FUNCTION_BLOCK AE_DEMUX_5 (* AE demultiplexor (generic FB) *)
  (* Standard: 61499-2; Description: Copyright (c) 2026 HR Agrartechnik GmbH This program and the accompanying materials are made available under the terms of the Eclipse Public License 2.0 which is available at https://www.eclipse.org/legal/epl-2.0/ SPDX-License-Identifier: EPL-2.0 *)
  (* Version 1.0, 2026-05-28, Franz Höpfinger, HR Agrartechnik GmbH *)
  PACKAGE adapter::selection::unidirectional;
  IMPORT eclipse4diac::core::TypeHash;
  {SET_ATTRIBUTE(eclipse4diac::core::GenericClassName, 'GEN_AE_DEMUX')}
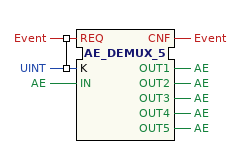
  EVENT_INPUT
    REQ WITH K; (* Set Index K *)
  END_EVENT
  EVENT_OUTPUT
    CNF; (* Confirmation of Set Index K *)
  END_EVENT
  VAR_INPUT
    K : UINT; (* index *)
  END_VAR
  SOCKETS
    IN : adapter::types::unidirectional::AE; (* Input Value to demultiplex *)
  END_SOCKETS
  PLUGS
    OUT1 : adapter::types::unidirectional::AE;
    OUT2 : adapter::types::unidirectional::AE;
    OUT3 : adapter::types::unidirectional::AE;
    OUT4 : adapter::types::unidirectional::AE;
    OUT5 : adapter::types::unidirectional::AE;
  END_PLUGS
END_FUNCTION_BLOCK
